PROGRAM WebHmi
VAR
	watchDog1 : TON;
	watchDog2 : TON;
END_VAR

WatchDog();



hmi.Jog_Speed := Hmi_Web.Jog_Speed;

// Fx 馬達位置
Hmi_Web.Fx_Pos := Axis.Fx.fPos;
// FxA 測長盤
Hmi_Web.FxA_Ex_Pos := Axis.FxA_Exp_Pos;
// FxB 測長盤
Hmi_Web.FxB_Ex_Pos := Axis.FxB_Exp_Pos;
	
// FxA 油壓夾輪位置
Hmi_Web.FxA_H_Pos := GroupFx.FxA_Clamp_Pos;
// FxB 油壓夾輪位置
Hmi_Web.FxB_H_Pos := GroupFx.FxB_Clamp_Pos;

WebHmi.Homming();

// 坐標系傳輸
Hmi_Web.WCS_A := GroupA.RefPos;

Hmi_Web.WCS_B := GroupB.RefPos;

Hmi_Web.WCS_C := GroupC.RefPos;

Hmi_Web.WCS_D := GroupD.RefPos;

ACTION Clamp:

END_ACTION

ACTION ErrorReset:
IF hmi.SysErrorRest THEN
	Safety.SystemError := FALSE;
	hmi.SysErrorRest := FALSE;
END_IF
END_ACTION

ACTION Homming:
IF Hmi_Web.Auto_homming THEN
	AutoMain.Homming();
	Hmi_Web.Auto_homming := FALSE;
END_IF
END_ACTION

ACTION WatchDog:
watchDog1(IN := NOT watchDog2.Q, PT:= T#500MS);
watchDog2(IN := watchDog1.Q, PT:= T#500MS);

Hmi_Web.Watchdog_Out := watchDog1.q;
END_ACTION

END_PROGRAM

(* stored: Version 1.1.0.1, ProductVersion 3.1.4026.13
   POU WebHmi: Id {7d27227b-25bd-493c-af6d-5b01257b715e}, SpecialFunc None
   Action Clamp: Id {6e3df157-7972-4f49-b719-7172aaa8a34f}
   Action ErrorReset: Id {49bf0790-ff85-4898-8789-5b6f95170134}
   Action Homming: Id {6f9c74fc-01de-4190-aafa-fa4fa76aae74}
   Action WatchDog: Id {8d35982f-38a0-4f62-af87-136a45b979d4} *)
